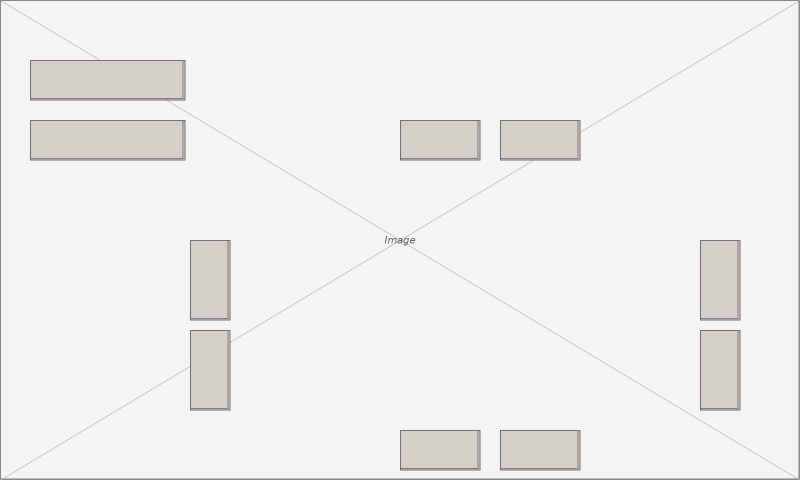
VISUALIZATION manualMode  // 800x480
    Image (0,0 800x480)
        p84334746: MAIN.bmpID
    Button (30,60 155x40), image: Buttons.homeButton
        OnMouseDown: change screen: Main
        OnMouseDown: execute { MAIN.manualModeON:=FALSE; }
    Button (30,120 155x40), image: Buttons.startButton
        OnMouseDown: toggle MAIN.manualModeON
    Button (190,330 40x80), invisible if: MAIN.caseImageUpdate.btn7, input disabled if: MAIN.caseImageUpdate.btn8, image: Buttons.down
        OnMouseClick: execute { Main.stateVar := 8; }
    Button (190,240 40x80), invisible if: MAIN.caseImageUpdate.btn8, input disabled if: MAIN.caseImageUpdate.btn8, image: Buttons.up
        OnMouseClick: execute { Main.stateVar := 1; }
    Button (700,240 40x80), invisible if: MAIN.caseImageUpdate.btn3, input disabled if: MAIN.caseImageUpdate.btn3, image: Buttons.up
        OnMouseClick: execute { Main.stateVar := 4; }
    Button (700,330 40x80), invisible if: MAIN.caseImageUpdate.btn4, input disabled if: MAIN.caseImageUpdate.btn4, image: Buttons.down
        OnMouseClick: execute { Main.stateVar := 5; }
    Button (500,430 80x40), invisible if: MAIN.caseImageUpdate.btn5, input disabled if: MAIN.caseImageUpdate.btn5, image: Buttons.right
        OnMouseClick: execute {
            IF MAIN.manualMode.prevState = 8 THEN
            	Main.stateVar := 7;
            END_IF
            IF MAIN.manualMode.prevState = 7 THEN
            	Main.stateVar := 6;
            END_IF
            IF MAIN.manualMode.prevState = 6 THEN
            	Main.stateVar := 5;
            END_IF
        }
    Button (400,430 80x40), invisible if: MAIN.caseImageUpdate.btn6, input disabled if: MAIN.caseImageUpdate.btn6, image: Buttons.left
        OnMouseClick: execute {
            IF MAIN.manualMode.prevState = 5 THEN
            	Main.stateVar := 6;
            END_IF
            IF MAIN.manualMode.prevState = 6 THEN
            	Main.stateVar := 7;
            END_IF
            IF MAIN.manualMode.prevState = 7 THEN
            	Main.stateVar := 8;
            END_IF
        }
    Button (400,120 80x40), invisible if: MAIN.caseImageUpdate.btn1, input disabled if: MAIN.caseImageUpdate.btn1, image: Buttons.left
        OnMouseClick: execute {
            IF MAIN.manualMode.prevState = 2 THEN
            	Main.stateVar := 1;
            END_IF
            IF MAIN.manualMode.prevState = 3 THEN
            	Main.stateVar := 2;
            END_IF
            IF MAIN.manualMode.prevState = 4 THEN
            	Main.stateVar := 3;
            END_IF
        }
    Button (500,120 80x40), invisible if: MAIN.caseImageUpdate.btn2, input disabled if: MAIN.caseImageUpdate.btn2, image: Buttons.right
        OnMouseClick: execute {
            IF MAIN.manualMode.prevState = 1 THEN
            	Main.stateVar := 2;
            END_IF
            IF MAIN.manualMode.prevState = 2 THEN
            	Main.stateVar := 3;
            END_IF
            IF MAIN.manualMode.prevState = 3 THEN
            	Main.stateVar := 4;
            END_IF
        }
END_VISUALIZATION

(* stored: Version 1.1.0.1, ProductVersion 3.1.4018.2
   Visu manualMode: Id {db7aafb4-62da-4faf-a749-9596ebb6025f} *)
